(* Logix 5000 project; controller Carpenter_Meter_SCP vendor 1 type 14 code 217 rev 31.11; software revision 31.01; part 5 of 7 *)
(* tags used below, declared in another part *)
   Carpenter_to_Pawnee_OK : BOOL;   // Carpenter to Pawnee Flow Path Permissive
   CC_HI_8800 : BOOL;   // Meter Skid MS-8800 Intrusion Deactivate Switch to OCC
   CC_HI_8840 : BOOL;   // Meter Skid MS-8840 Intrusion Deactivate Switch to OCC
   CC_OCC_HB : DINT;   // Heartbeat from OCC to SCP
   CC_PI_1101 : OCC_Analog;   // Station Discharge Pressure to OCC
   CC_SCP_HB : DINT;   // Heartbeat from SCP to OCC
   CC_XA_0020A : BOOL;   // SCP Main Panel 24VDC Fail to OCC
   CC_XA_0021A : BOOL;   // FGP Main Panel 24VDC Fail to OCC
   CC_XI_0001 : BOOL;   // QA Building Intrusion Deactivate Switch to OCC
   CC_XI_0001A : BOOL;   // QA Building Intrusion Switch to OCC
   CC_XI_0011A : BOOL;   // PDC Building Intrusion Switch to OCC
   CC_XI_0011B : BOOL;   // PDC Building Intrusion Deactivate Switch to OCC
   CC_XI_0020 : BOOL;   // SCP Main PLC 24VDC Failure to OCC
   CC_XI_8800 : BOOL;   // Meter Skid MS-8800 Intrusion Switch to OCC
   CC_XI_8800A : BOOL;   // MS8800 SCP 24VDC Failure to OCC
   CC_XI_8840 : BOOL;   // Meter Skid MS-8840 Intrusion Switch to OCC
   CC_XI_8840A : BOOL;   // MS8840 SCP 24VDC Failure to OCC
   CC_ZI_1100A : BOOL;   // Pig Launched Pig Sig to OCC
   CC_ZI_1100B : BOOL;   // Pig Station Depart Pig Sig to OCC
   CCS_AI_0001 : OCC_Analog;   // QA Building Gas Detector to OCC (AIT-0001)
   CCS_AI_8800A : OCC_Analog;   // Meter Skid MS-8800 Gas Detector #1 (AIT-8800A)
   CCS_AI_8800B : OCC_Analog;   // Meter Skid MS-8800 Gas Detector #2 (AIT-8800B)
   CCS_AI_8840A : OCC_Analog;   // Meter Skid MS-8840 Gas Detector #1 (AIT-8840A)
   CCS_AI_8840B : OCC_Analog;   // Meter Skid MS-8840 Gas Detector #2 (AIT-8840B)
   CCS_ESD_Active : BOOL;   // Station ESD Active to OCC
   CCS_ESD_OCC : BOOL;   // Station ESD Command from OCC
   CCS_FGP_Deactivate : BOOL;   // Fire and Gas Deactivated Status to OCC
   CCS_HI_0011A : BOOL;   // PDC ESD Pushbutton to OCC
   CCS_HI_0017 : BOOL;   // PDC Building PLC Panel ESD Pushbutton to OCC
   CCS_HI_0112A : BOOL;   // QA Building ESD Pushbutton #1 to OCC
   CCS_HI_0112B : BOOL;   // QA Building ESD Pushbutton #2 to OCC
   CCS_HI_0113 : BOOL;   // South Gate ESD Pushbutton to OCC
   CCS_HI_0114 : BOOL;   // North Gate ESD Pushbutton to OCC
   CCS_HI_8800A : BOOL;   // Meter Skid MS-8800 ESD Pushbutton #1 to OCC
   CCS_HI_8800B : BOOL;   // Meter Skid MS-8800 ESD Pushbutton #2 to OCC
   CCS_HI_8840A : BOOL;   // Meter Skid MS-8840 ESD Pushbutton #1 to OCC
   CCS_HI_8840B : BOOL;   // Meter Skid MS-8840 ESD Pushbutton #1 to OCC
   CCS_LAH_3000 : BOOL;   // Sump Tank TU-3000 Leak Detection Switch to OCC
   CCS_LAH_3000_inhibit : BOOL;   // Sump Tank TU-3000 Leak Detection Switch Inhibited to OCC
   CCS_LAH_3100 : BOOL;   // Sump Tank TU-3100 Leak Detection Switch to OCC
   CCS_LAH_3100_inhibit : BOOL;   // Sump Tank TU-3100 Leak Detection Switch Inhibited to OCC
   CCS_LAHH_3000 : BOOL;   // Sump Tank TU-3000 HiHi Level Switch to OCC
   CCS_LAHH_3000_inhibit : BOOL;   // Sump Tank TU-3000 HiHi Level Switch Inhibited to OCC
   CCS_LAHH_3100 : BOOL;   // Sump Tank TU-3100 HiHi Level Switch to OCC
   CCS_LAHH_3100_inhibit : BOOL;   // Sump Tank TU-3100 HiHi Level Switch inhibited to OCC
   CCS_LI_3000 : OCC_Analog;   // Sump Tank TU-3000 Level to OCC
   CCS_LI_3100 : OCC_Analog;   // Sump Tank TU-3000 Level to OCC
   CCS_TI_8010 : OCC_Analog;   // PDC Building Temperature (TIT-8010)
   CCS_XI_0029A : BOOL;   // QA Building Smoke Detector #1 to OCC
   CCS_XI_0029A_Inhibit : BOOL;   // QA Building Smoke Detector #1 Inhibit to OCC
   CCS_XI_0029B : BOOL;   // QA Building Smoke Detector #2 to OCC
   CCS_XI_0029B_Inhibit : BOOL;   // QA Building Smoke Detector #2 Inhibit to OCC
   CCS_XV_0001 : BaseVLVLiquid;   // XV-0001 OCC
   CCS_XV_0041 : BaseVLVLiquid;   // XV-0041 OCC
   CCS_XV_1100 : BaseVLVLiquid;   // XV-1100 OCC
   CCS_XV_1101 : BaseVLVLiquid;   // XV-1101 OCC
   CCS_YI_0022A : BOOL;   // PDC Smoke Detector to OCC
   CCS_YI_0022A_Inhibit : BOOL;   // PDC Smoke Detector Inhibit to OCC
   Cust1_WIOM_Alarm : BOOL;   // Customer 1 WIOM Alarm
   Customer1_Flowpath_OK : BOOL;   // Customer #1 Flowpath Permissive (1 = OK)
   Customer5_Flowpath_OK : BOOL;   // Customer #5 Flowpath Permissive (1 = OK)
   fgp_deactivate_keysw : BOOL;   // Fire and Gas System Deactivated through Key Switch
   FGP_ESD : TGE_Alarm;   // ESD Shutdown from FGP (HS-0020A)
   FGP_Produced : BasProdCons;   // FGP Produced Data
   FGP_SCADA : BasProdCons;
   FI_8800 : REAL;   // Meter Skid MS-8800 Flow Rate in GSV from EFM
   FI_8840 : REAL;   // Meter Skid MS-8840 Flow Rate from EFM
   hb_fail_scada : BOOL;   // SCADA HB Failure
   hb_timer_scada : TIMER;   // SCADA HB Timer
   Launcher_Pig_Sig : TGE_Alarm;   // Launcher Pig Signal (ZS-1100A)
   Main_FGP_24VDC_Fail : TGE_Alarm;   // Main PLC FGP 24VDC Fail (XS-0021)
   MS8800_Biocide_BBL_Per_Day : REAL;   // MS8800 Biocide Flow Rate in BBL/Day (Based off set target of 500PPM)
   MS8800_Biocide_Flow_SP : REAL;   // Meter Skid MS-8800 Biocide Flow Rate Gal/Day
   MS8800_Biocide_RunReq : BOOL;   // Meter Skid MS8800 Biocide Run Req
   MS8800_Cust_Press : TGE_AI_UDT;   // Meter Skid MS-8800 Customer Inlet Pressure (Communicated from Cust)
   MS8800_Flow_Control : PID;   // Meter Skid MS8800 Flow Rate P&ID
   MS8800_Inlet_Press_Control : PID;   // Meter Skid MS8800 Customer Inlet Pressure P&ID
   MS8800_Intrusion : IntrusionAlm;   // Meter Skid MS-8800 Intrusion #1 Alarm
   MS8800_OilFlow_BBL_Per_Day : REAL;   // Meter Skid MS-8800 Oil Flow Rate in BBL/Day
   MS8800_PCV_Pos_AOI : TGE_AI;   // Meter Skid MS-8800 Pressure Control Valve - Position Feedback (PCV-0001)
   MS8800_WaterFlow_BBL_Per_Day : REAL;   // MS8800 Water Flow Rate in BBL/Day (Based off 1% oil in water)
   MS8840_Biocide_BBL_Per_Day : REAL;   // MS8840 Biocide Flow Rate in BBL/Day (Based off set target of 500PPM)
   MS8840_Biocide_Flow_SP : REAL;   // Meter Skid MS-8840 Biocide Flow Rate Gal/Day
   MS8840_Biocide_RunReq : BOOL;   // Meter Skid MS8840 Biocide Run Req
   MS8840_Cust_Press : TGE_AI_UDT;   // Meter Skid MS-8840 Customer Inlet Pressure (Communicated from Cust)
   MS8840_Flow_Control : PID;   // Meter Skid MS8840 Flow Rate P&ID
   MS8840_Inlet_Press_Control : PID;   // Meter Skid MS8840 Customer Inlet Pressure P&ID
   MS8840_Intrusion : IntrusionAlm;   // Meter Skid MS-8840 Intrusion Alarm
   MS8840_OilFlow_BBL_Per_Day : REAL;   // Meter Skid MS-8840 Oil Flow Rate in BBL/Day
   MS8840_PCV_Pos_AOI : TGE_AI;   // Meter Skid MS-8840 Pressure Control Valve - Position Feedback (PCV-0041)
   MS8840_WaterFlow_BBL_Per_Day : REAL;   // MS8840 Water Flow Rate in BBL/Day (Based off 1% oil in water)
   OCC_hb_old : DINT;   // Old OCC HB for diagnostic purposes
   PDC_Bldg_Intrusion : IntrusionAlm;   // PDC Building Intrusion Alarm
   PIC_0001A_Out : REAL;   // Control Valve Output Variable Related to Inlet Pressure
   PIC_0001B_Out : REAL;   // Control Valve Ouptut Variable related to Flow Rate
   PIC_0041A_Out : REAL;   // Control Valve Output Variable Related to Inlet Pressure
   PIC_0041B_Out : REAL;   // Control Valve Ouptut Variable related to Flow Rate
   PV0001_Error : REAL;   // PV0001 Command vs. Feedback Error
   PV0001_Malf : TGE_Alarm;   // PV0001 Malfunction Alarm
   PV0001_Pos_Cmd : REAL;   // PCV-0001 Position Command
   PV0041_Error : REAL;   // PV0041 Command vs. Feedback Error
   PV0041_Malf : TGE_Alarm;   // PV0041 Malfunction Alarm
   PV0041_Pos_Cmd : REAL;   // PCV-0041 Position Command
   pv_0001_pid_tmr : TIMER;
   pv_0041_pid_tmr : TIMER;
   QA_Bldg_Intrusion : IntrusionAlm;   // QA Building Intrusion Alarm Bit 0-7 = Bldg Int Switch Bit 15 = Deact HS
   SCP_Produced : BasProdCons;
   Sta_Stat : StaStatus;
   sta_stop_vlv_req : BOOL;   // Station Stop Valve Close Request
   Station_Depart_Pig_Sig : TGE_Alarm;   // Station Departed Pig Signal (ZS-1100B)
   Station_Disch_Press : TGE_AI_UDT;   // Station Discharge Pressure - Launcher Skid (PIT-1101)
   TU3000_HiHi_Lvl : TGE_Alarm;   // Sump Tank (TU-3000) Hi Hi Level Switch (LSHH-3000)
   TU3000_Leak_Detect : TGE_Alarm;   // Sump Tank (TU-3000) Leak Detected (LSH-3000)
   TU3000_Level : TGE_AI_UDT;   // Sump Tank (TU-3000) Level Transmitter (LIT-3000)
   TU3100_HiHi_Lvl : TGE_Alarm;   // Sump Tank (TU-3100) Hi Hi Level Switch (LSHH-3100)
   TU3100_Leak_Detect : TGE_Alarm;   // Sump Tank (TU-3100) Leak Detected (LSH-3100)
   TU3100_Level : TGE_AI_UDT;   // Sump Tank (TU-3100) Level Transmitter (LIT-3100)
   watchdog_tmr : TIMER;   // Watchdog Timer for Communications
   XV_0001 : BaseVLVLiquid;   // XV-0001
   XV_0041 : BaseVLVLiquid;   // XV-0041
   XV_1100 : BaseVLVLiquid;   // XV-1100
   XV_1101 : BaseVLVLiquid;   // XV-1101
(* Map_Inputs, continued *)

ROUTINE Main   (* ladder *)
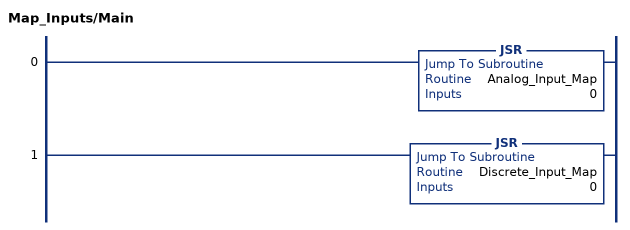
   0: JSR(Analog_Input_Map,0);
   1: JSR(Discrete_Input_Map,0);
END_ROUTINE
END_PROGRAM

PROGRAM Map_Outputs   (* main routine Main *)

ROUTINE Analog_Output_Map   (* ladder *)
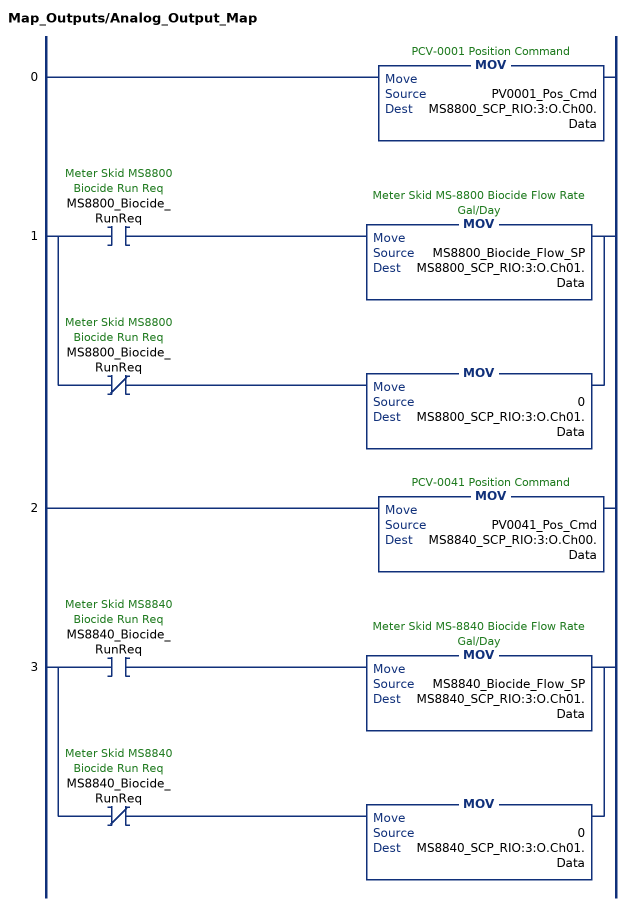
   0: MOV(PV0001_Pos_Cmd,MS8800_SCP_RIO:3:O.Ch00.Data);
   1: [XIC(MS8800_Biocide_RunReq) MOV(MS8800_Biocide_Flow_SP,MS8800_SCP_RIO:3:O.Ch01.Data) ,XIO(MS8800_Biocide_RunReq) MOV(0,MS8800_SCP_RIO:3:O.Ch01.Data) ];
   2: MOV(PV0041_Pos_Cmd,MS8840_SCP_RIO:3:O.Ch00.Data);
   3: [XIC(MS8840_Biocide_RunReq) MOV(MS8840_Biocide_Flow_SP,MS8840_SCP_RIO:3:O.Ch01.Data) ,XIO(MS8840_Biocide_RunReq) MOV(0,MS8840_SCP_RIO:3:O.Ch01.Data) ];
END_ROUTINE

ROUTINE Discrete_Output_Map   (* ladder *)
   0: NOP();
END_ROUTINE

ROUTINE Main   (* ladder *)
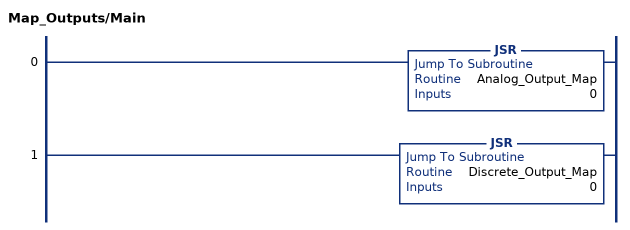
   0: JSR(Analog_Output_Map,0);
   1: JSR(Discrete_Output_Map,0);
END_ROUTINE
END_PROGRAM

PROGRAM Meter_Skid_Control   (* main routine Main *)

ROUTINE Main   (* ladder *)
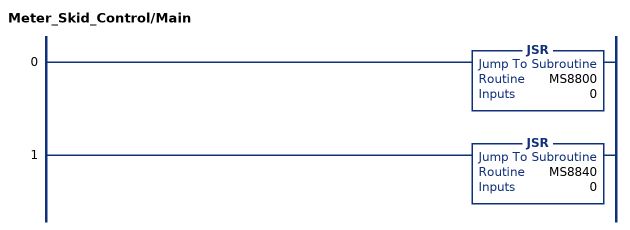
   0: JSR(MS8800,0);
   1: JSR(MS8840,0);
END_ROUTINE

ROUTINE MS8800   (* ladder *)
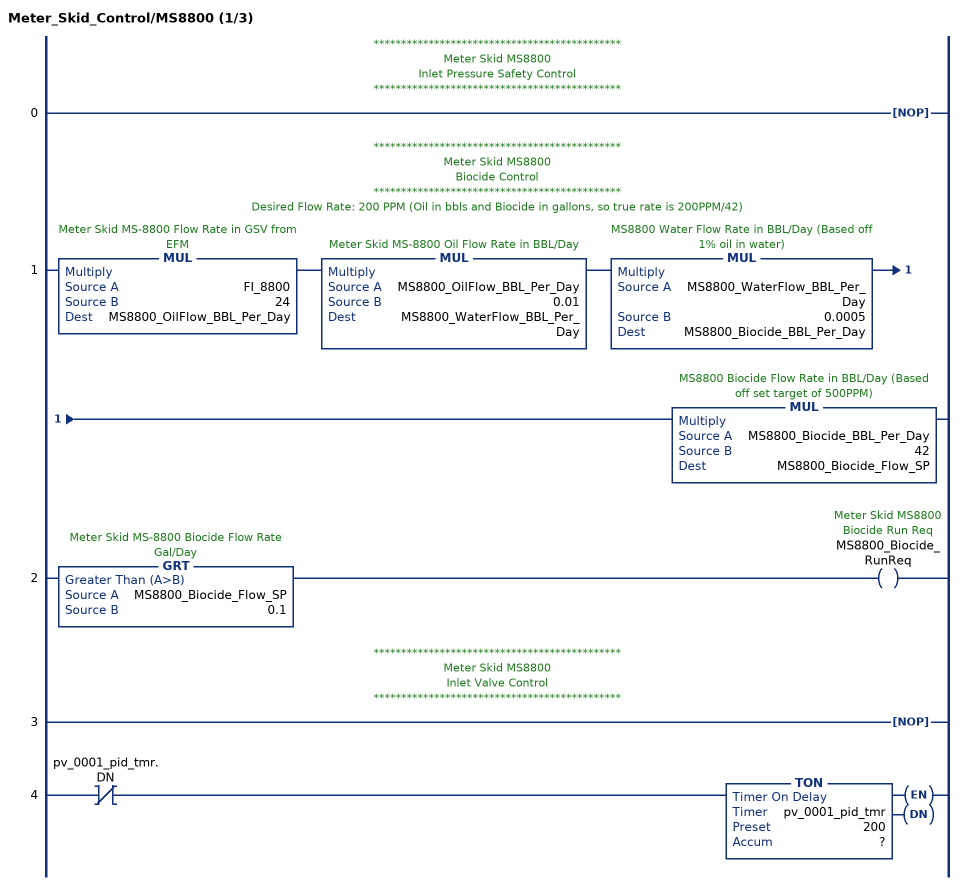
   // *********************************************
   // Meter Skid MS8800
   // Inlet Pressure Safety Control
   // *********************************************
   0: NOP();
   // *********************************************
   // Meter Skid MS8800
   // Biocide Control
   // *********************************************
   // Desired Flow Rate: 200 PPM (Oil in bbls and Biocide in gallons, so true rate is 200PPM/42)
   1: MUL(FI_8800,24,MS8800_OilFlow_BBL_Per_Day)MUL(MS8800_OilFlow_BBL_Per_Day,0.01,MS8800_WaterFlow_BBL_Per_Day)MUL(MS8800_WaterFlow_BBL_Per_Day,0.0005,MS8800_Biocide_BBL_Per_Day)MUL(MS8800_Biocide_BBL_Per_Day,42,MS8800_Biocide_Flow_SP);
   2: GRT(MS8800_Biocide_Flow_SP,0.1)OTE(MS8800_Biocide_RunReq);
   // *********************************************
   // Meter Skid MS8800
   // Inlet Valve Control
   // *********************************************
   3: NOP();
   4: XIO(pv_0001_pid_tmr.DN)TON(pv_0001_pid_tmr,?,?);
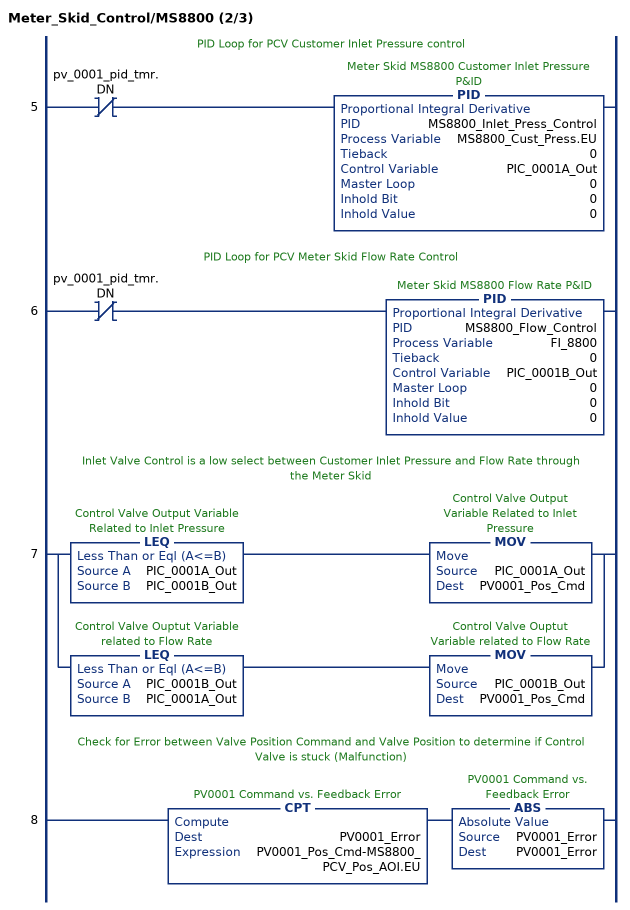
   // PID Loop for PCV Customer Inlet Pressure control
   5: XIO(pv_0001_pid_tmr.DN)PID(MS8800_Inlet_Press_Control,MS8800_Cust_Press.EU,0,PIC_0001A_Out,0,0,0);
   // PID Loop for PCV Meter Skid Flow Rate Control
   6: XIO(pv_0001_pid_tmr.DN)PID(MS8800_Flow_Control,FI_8800,0,PIC_0001B_Out,0,0,0);
   // Inlet Valve Control is a low select between Customer Inlet Pressure and Flow Rate through the Meter Skid
   7: [LEQ(PIC_0001A_Out,PIC_0001B_Out) MOV(PIC_0001A_Out,PV0001_Pos_Cmd) ,LEQ(PIC_0001B_Out,PIC_0001A_Out) MOV(PIC_0001B_Out,PV0001_Pos_Cmd) ];
   // Check for Error between Valve Position Command and Valve Position to determine if Control Valve is stuck (Malfunction)
   8: CPT(PV0001_Error,PV0001_Pos_Cmd-MS8800_PCV_Pos_AOI.EU)ABS(PV0001_Error,PV0001_Error);
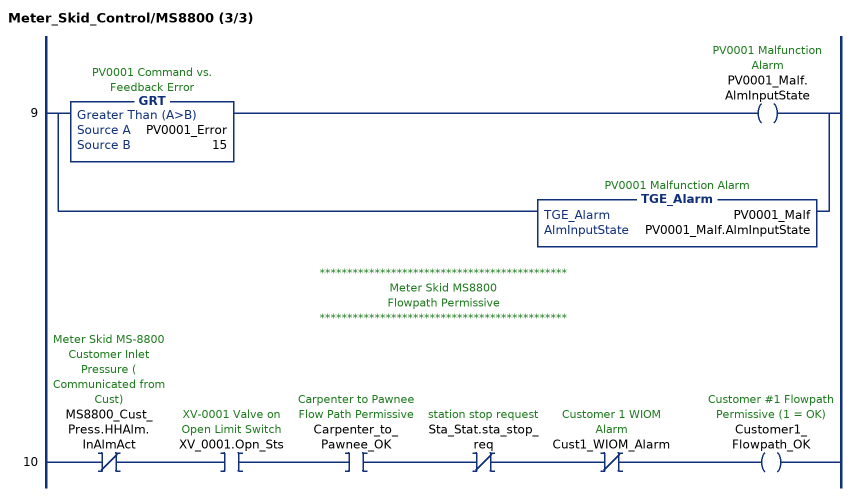
   9: [GRT(PV0001_Error,15) OTE(PV0001_Malf.AlmInputState) ,TGE_Alarm(PV0001_Malf,PV0001_Malf.AlmInputState) ];
   // *********************************************
   // Meter Skid MS8800
   // Flowpath Permissive
   // *********************************************
   10: XIO(MS8800_Cust_Press.HHAlm.InAlmAct)XIC(XV_0001.Opn_Sts)XIC(Carpenter_to_Pawnee_OK)XIO(Sta_Stat.sta_stop_req)XIO(Cust1_WIOM_Alarm)OTE(Customer1_Flowpath_OK);
END_ROUTINE

ROUTINE MS8840   (* ladder *)
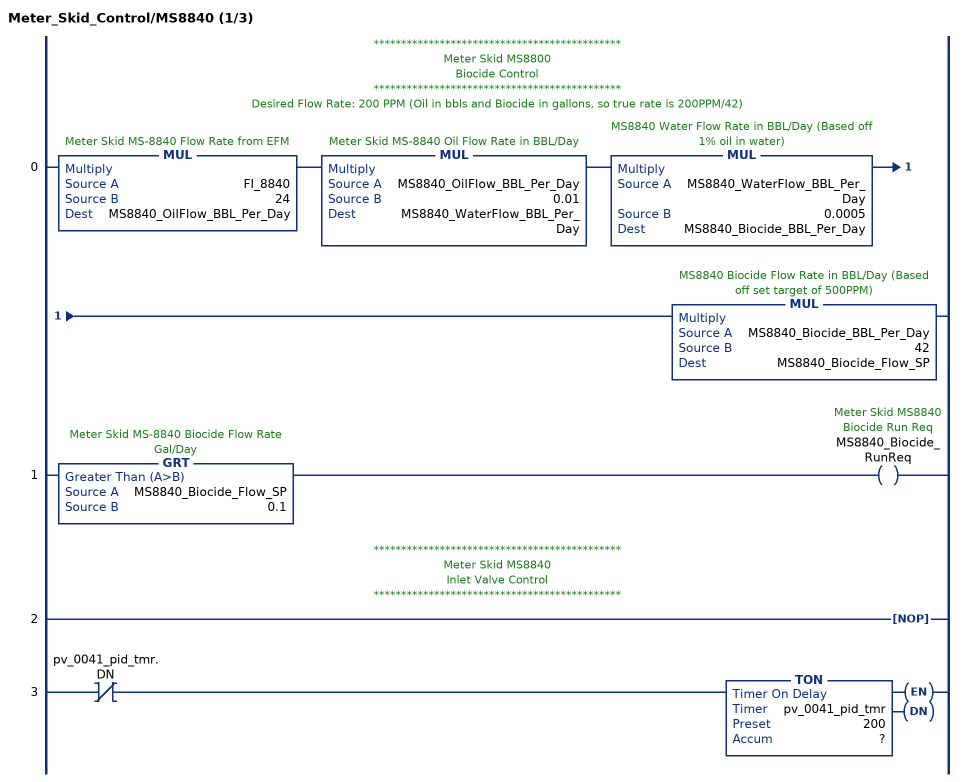
   // *********************************************
   // Meter Skid MS8800
   // Biocide Control
   // *********************************************
   // Desired Flow Rate: 200 PPM (Oil in bbls and Biocide in gallons, so true rate is 200PPM/42)
   0: MUL(FI_8840,24,MS8840_OilFlow_BBL_Per_Day)MUL(MS8840_OilFlow_BBL_Per_Day,0.01,MS8840_WaterFlow_BBL_Per_Day)MUL(MS8840_WaterFlow_BBL_Per_Day,0.0005,MS8840_Biocide_BBL_Per_Day)MUL(MS8840_Biocide_BBL_Per_Day,42,MS8840_Biocide_Flow_SP);
   1: GRT(MS8840_Biocide_Flow_SP,0.1)OTE(MS8840_Biocide_RunReq);
   // *********************************************
   // Meter Skid MS8840
   // Inlet Valve Control
   // *********************************************
   2: NOP();
   3: XIO(pv_0041_pid_tmr.DN)TON(pv_0041_pid_tmr,?,?);
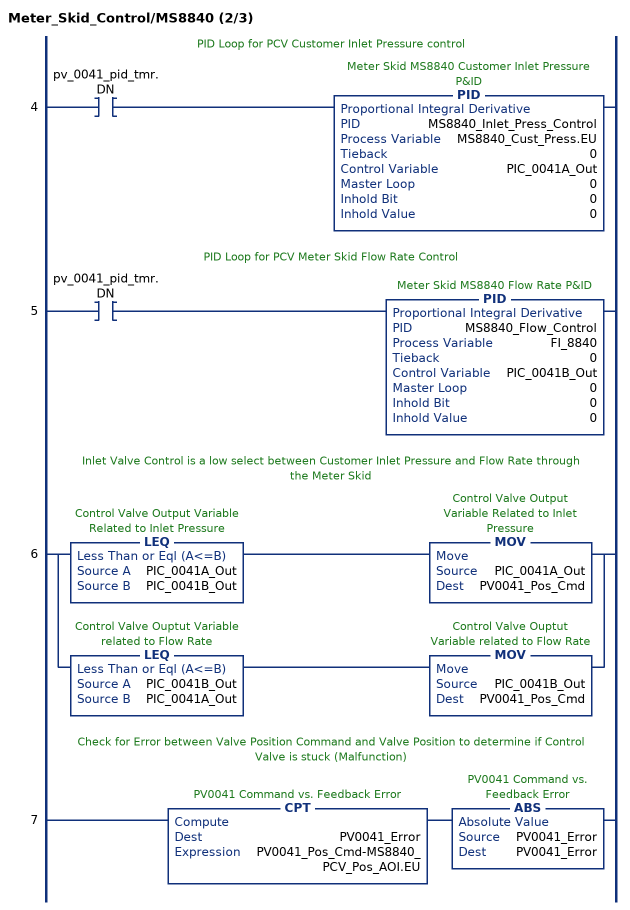
   // PID Loop for PCV Customer Inlet Pressure control
   4: XIC(pv_0041_pid_tmr.DN)PID(MS8840_Inlet_Press_Control,MS8840_Cust_Press.EU,0,PIC_0041A_Out,0,0,0);
   // PID Loop for PCV Meter Skid Flow Rate Control
   5: XIC(pv_0041_pid_tmr.DN)PID(MS8840_Flow_Control,FI_8840,0,PIC_0041B_Out,0,0,0);
   // Inlet Valve Control is a low select between Customer Inlet Pressure and Flow Rate through the Meter Skid
   6: [LEQ(PIC_0041A_Out,PIC_0041B_Out) MOV(PIC_0041A_Out,PV0041_Pos_Cmd) ,LEQ(PIC_0041B_Out,PIC_0041A_Out) MOV(PIC_0041B_Out,PV0041_Pos_Cmd) ];
   // Check for Error between Valve Position Command and Valve Position to determine if Control Valve is stuck (Malfunction)
   7: CPT(PV0041_Error,PV0041_Pos_Cmd-MS8840_PCV_Pos_AOI.EU)ABS(PV0041_Error,PV0041_Error);
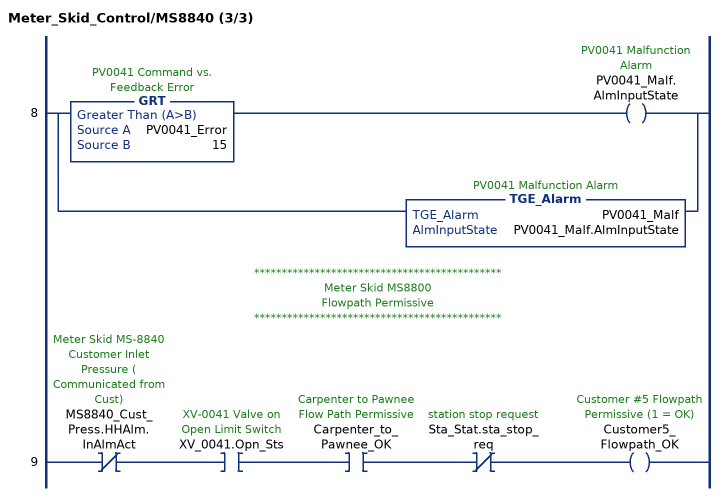
   8: [GRT(PV0041_Error,15) OTE(PV0041_Malf.AlmInputState) ,TGE_Alarm(PV0041_Malf,PV0041_Malf.AlmInputState) ];
   // *********************************************
   // Meter Skid MS8800
   // Flowpath Permissive
   // *********************************************
   9: XIO(MS8840_Cust_Press.HHAlm.InAlmAct)XIC(XV_0041.Opn_Sts)XIC(Carpenter_to_Pawnee_OK)XIO(Sta_Stat.sta_stop_req)OTE(Customer5_Flowpath_OK);
END_ROUTINE
END_PROGRAM

PROGRAM OCC_Comms   (* main routine OCC_Comms_Main *)

ROUTINE OCC_Comms_Main   (* ladder *)
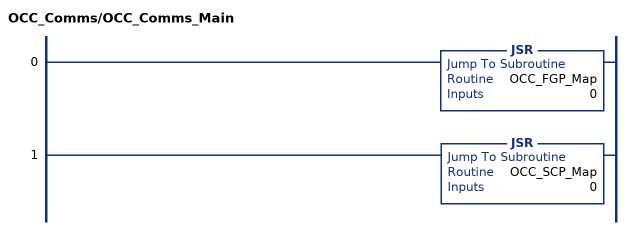
   0: JSR(OCC_FGP_Map,0);
   1: JSR(OCC_SCP_Map,0);
END_ROUTINE

ROUTINE OCC_FGP_Map   (* ladder *)
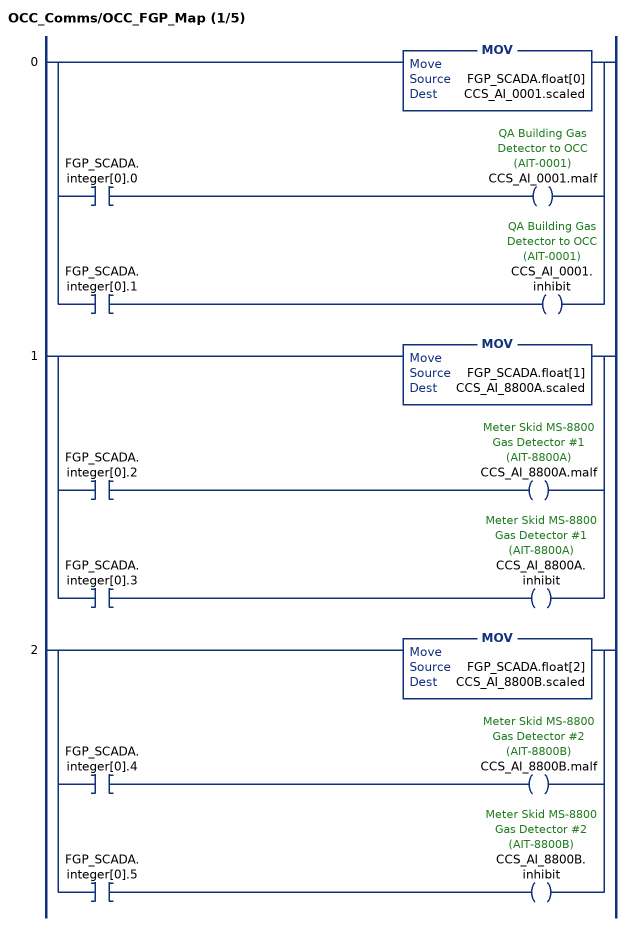
   0: [MOV(FGP_SCADA.float[0],CCS_AI_0001.scaled) ,XIC(FGP_SCADA.integer[0].0) OTE(CCS_AI_0001.malf) ,XIC(FGP_SCADA.integer[0].1) OTE(CCS_AI_0001.inhibit) ];
   1: [MOV(FGP_SCADA.float[1],CCS_AI_8800A.scaled) ,XIC(FGP_SCADA.integer[0].2) OTE(CCS_AI_8800A.malf) ,XIC(FGP_SCADA.integer[0].3) OTE(CCS_AI_8800A.inhibit) ];
   2: [MOV(FGP_SCADA.float[2],CCS_AI_8800B.scaled) ,XIC(FGP_SCADA.integer[0].4) OTE(CCS_AI_8800B.malf) ,XIC(FGP_SCADA.integer[0].5) OTE(CCS_AI_8800B.inhibit) ];
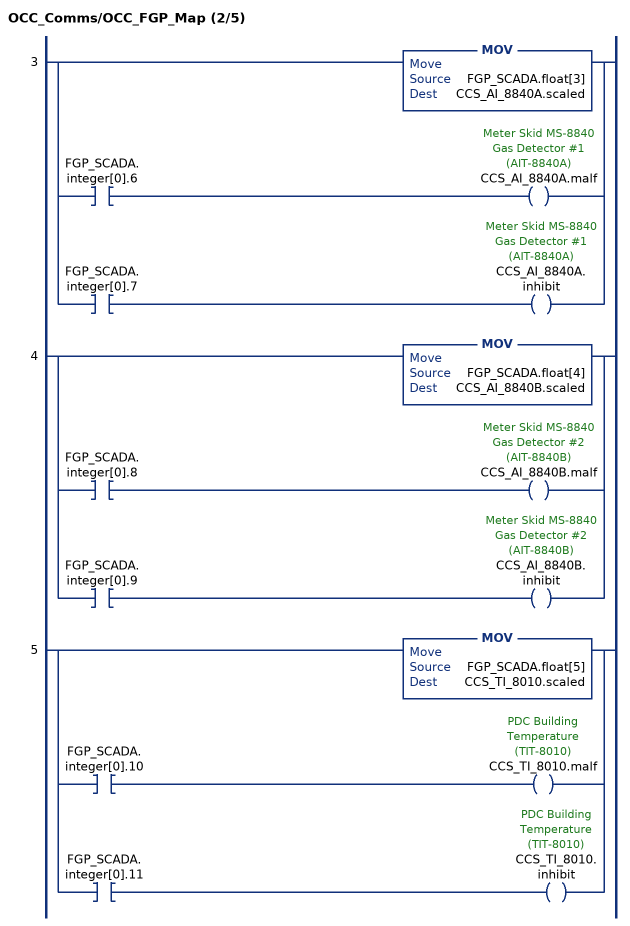
   3: [MOV(FGP_SCADA.float[3],CCS_AI_8840A.scaled) ,XIC(FGP_SCADA.integer[0].6) OTE(CCS_AI_8840A.malf) ,XIC(FGP_SCADA.integer[0].7) OTE(CCS_AI_8840A.inhibit) ];
   4: [MOV(FGP_SCADA.float[4],CCS_AI_8840B.scaled) ,XIC(FGP_SCADA.integer[0].8) OTE(CCS_AI_8840B.malf) ,XIC(FGP_SCADA.integer[0].9) OTE(CCS_AI_8840B.inhibit) ];
   5: [MOV(FGP_SCADA.float[5],CCS_TI_8010.scaled) ,XIC(FGP_SCADA.integer[0].10) OTE(CCS_TI_8010.malf) ,XIC(FGP_SCADA.integer[0].11) OTE(CCS_TI_8010.inhibit) ];
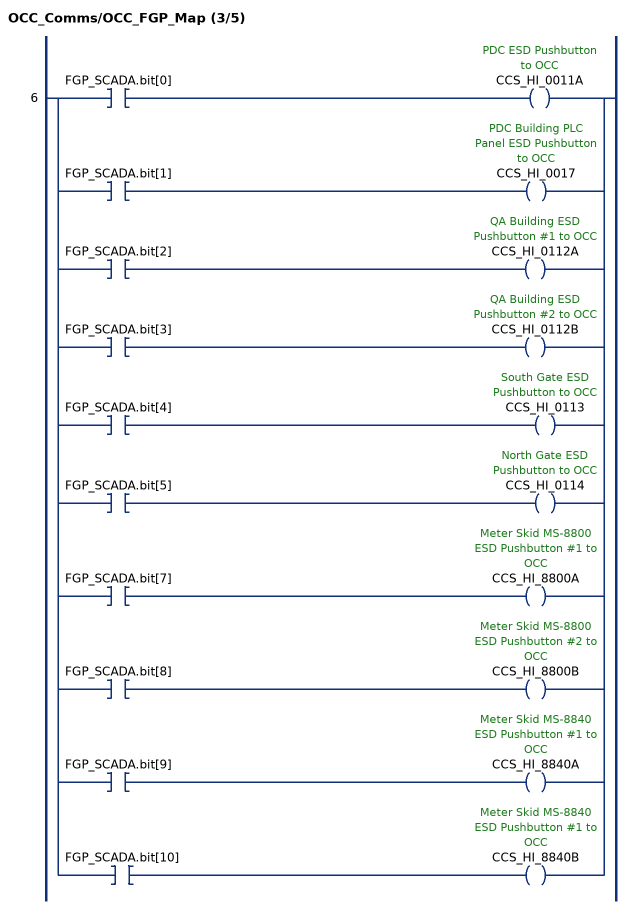
   6: [XIC(FGP_SCADA.bit[0]) OTE(CCS_HI_0011A) ,XIC(FGP_SCADA.bit[1]) OTE(CCS_HI_0017) ,XIC(FGP_SCADA.bit[2]) OTE(CCS_HI_0112A) ,XIC(FGP_SCADA.bit[3]) OTE(CCS_HI_0112B) ,XIC(FGP_SCADA.bit[4]) OTE(CCS_HI_0113) ,XIC(FGP_SCADA.bit[5]) OTE(CCS_HI_0114) ,XIC(FGP_SCADA.bit[7]) OTE(CCS_HI_8800A) ,XIC(FGP_SCADA.bit[8]) OTE(CCS_HI_8800B) ,XIC(FGP_SCADA.bit[9]) OTE(CCS_HI_8840A) ,XIC(FGP_SCADA.bit[10]) OTE(CCS_HI_8840B) ];
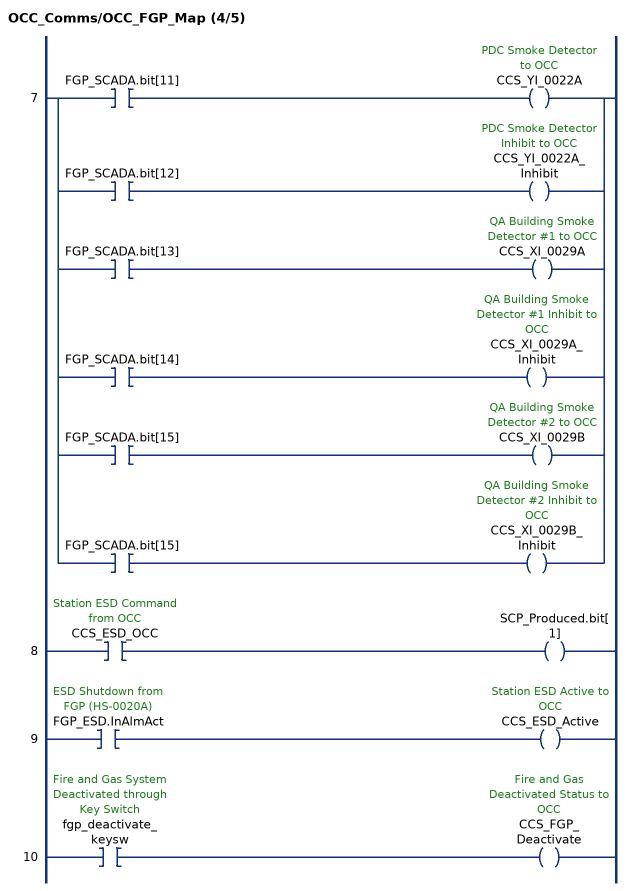
   7: [XIC(FGP_SCADA.bit[11]) OTE(CCS_YI_0022A) ,XIC(FGP_SCADA.bit[12]) OTE(CCS_YI_0022A_Inhibit) ,XIC(FGP_SCADA.bit[13]) OTE(CCS_XI_0029A) ,XIC(FGP_SCADA.bit[14]) OTE(CCS_XI_0029A_Inhibit) ,XIC(FGP_SCADA.bit[15]) OTE(CCS_XI_0029B) ,XIC(FGP_SCADA.bit[15]) OTE(CCS_XI_0029B_Inhibit) ];
   8: XIC(CCS_ESD_OCC)OTE(SCP_Produced.bit[1]);
   9: XIC(FGP_ESD.InAlmAct)OTE(CCS_ESD_Active);
   10: XIC(fgp_deactivate_keysw)OTE(CCS_FGP_Deactivate);
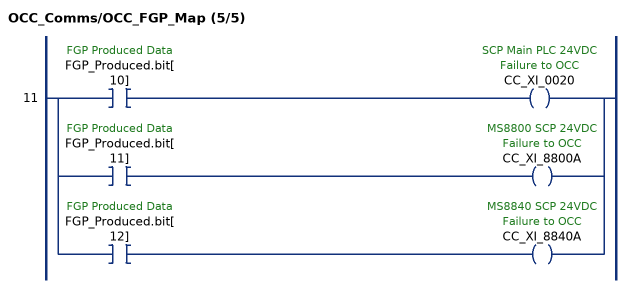
   11: [XIC(FGP_Produced.bit[10]) OTE(CC_XI_0020) ,XIC(FGP_Produced.bit[11]) OTE(CC_XI_8800A) ,XIC(FGP_Produced.bit[12]) OTE(CC_XI_8840A) ];
END_ROUTINE

ROUTINE OCC_SCP_Map   (* ladder *)
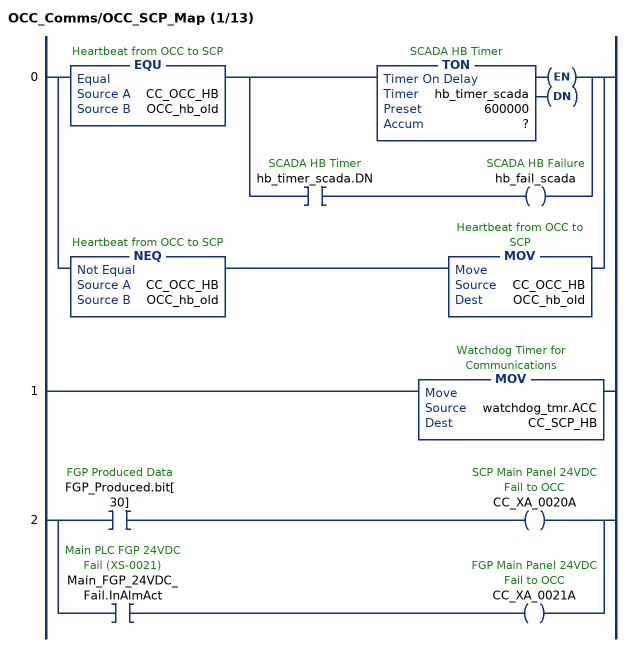
   0: [EQU(CC_OCC_HB,OCC_hb_old) [TON(hb_timer_scada,?,?) ,XIC(hb_timer_scada.DN) OTE(hb_fail_scada) ] ,NEQ(CC_OCC_HB,OCC_hb_old) MOV(CC_OCC_HB,OCC_hb_old) ];
   1: MOV(watchdog_tmr.ACC,CC_SCP_HB);
   2: [XIC(FGP_Produced.bit[30]) OTE(CC_XA_0020A) ,XIC(Main_FGP_24VDC_Fail.InAlmAct) OTE(CC_XA_0021A) ];
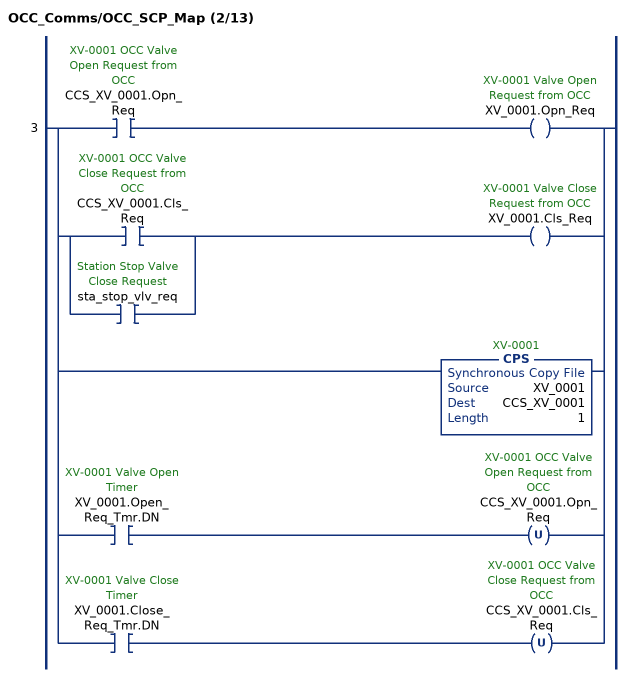
   3: [XIC(CCS_XV_0001.Opn_Req) OTE(XV_0001.Opn_Req) ,[XIC(CCS_XV_0001.Cls_Req) ,XIC(sta_stop_vlv_req) ] OTE(XV_0001.Cls_Req) ,CPS(XV_0001,CCS_XV_0001,1) ,XIC(XV_0001.Open_Req_Tmr.DN) OTU(CCS_XV_0001.Opn_Req) ,XIC(XV_0001.Close_Req_Tmr.DN) OTU(CCS_XV_0001.Cls_Req) ];
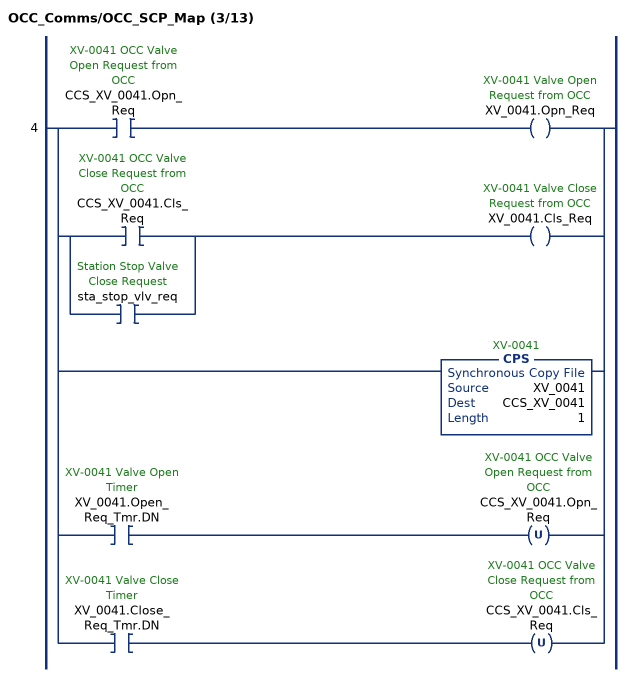
   4: [XIC(CCS_XV_0041.Opn_Req) OTE(XV_0041.Opn_Req) ,[XIC(CCS_XV_0041.Cls_Req) ,XIC(sta_stop_vlv_req) ] OTE(XV_0041.Cls_Req) ,CPS(XV_0041,CCS_XV_0041,1) ,XIC(XV_0041.Open_Req_Tmr.DN) OTU(CCS_XV_0041.Opn_Req) ,XIC(XV_0041.Close_Req_Tmr.DN) OTU(CCS_XV_0041.Cls_Req) ];
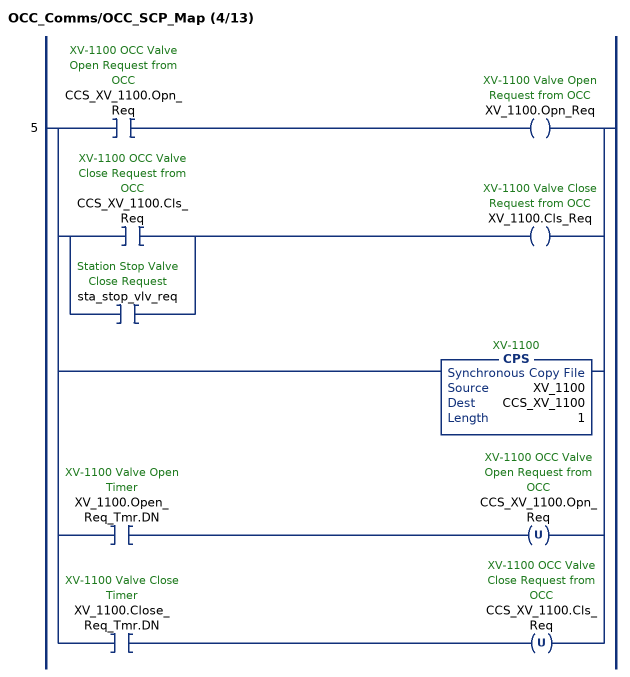
   5: [XIC(CCS_XV_1100.Opn_Req) OTE(XV_1100.Opn_Req) ,[XIC(CCS_XV_1100.Cls_Req) ,XIC(sta_stop_vlv_req) ] OTE(XV_1100.Cls_Req) ,CPS(XV_1100,CCS_XV_1100,1) ,XIC(XV_1100.Open_Req_Tmr.DN) OTU(CCS_XV_1100.Opn_Req) ,XIC(XV_1100.Close_Req_Tmr.DN) OTU(CCS_XV_1100.Cls_Req) ];
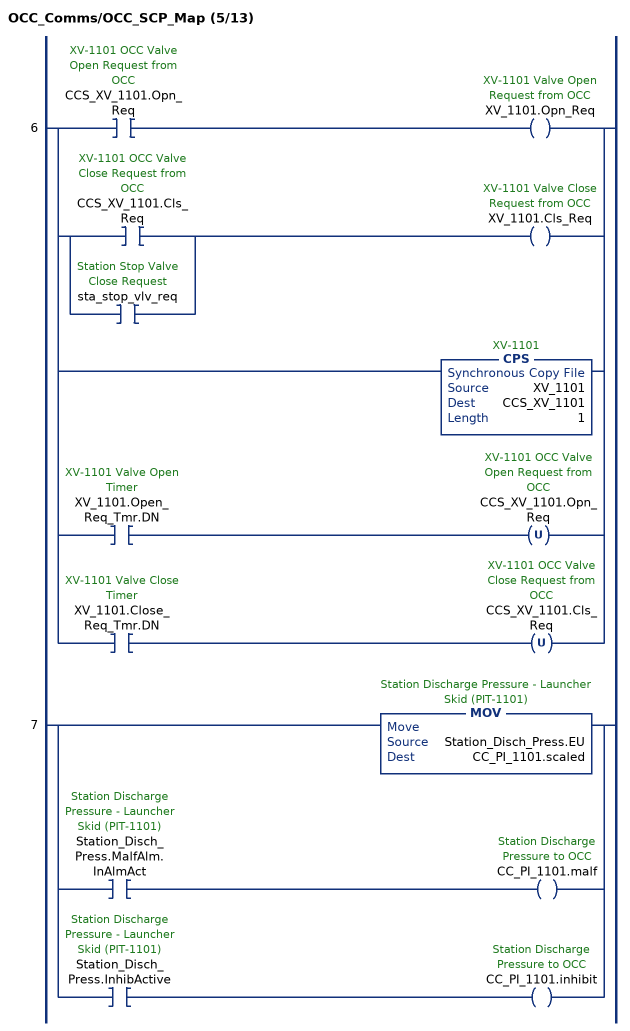
   6: [XIC(CCS_XV_1101.Opn_Req) OTE(XV_1101.Opn_Req) ,[XIC(CCS_XV_1101.Cls_Req) ,XIC(sta_stop_vlv_req) ] OTE(XV_1101.Cls_Req) ,CPS(XV_1101,CCS_XV_1101,1) ,XIC(XV_1101.Open_Req_Tmr.DN) OTU(CCS_XV_1101.Opn_Req) ,XIC(XV_1101.Close_Req_Tmr.DN) OTU(CCS_XV_1101.Cls_Req) ];
   7: [MOV(Station_Disch_Press.EU,CC_PI_1101.scaled) ,XIC(Station_Disch_Press.MalfAlm.InAlmAct) OTE(CC_PI_1101.malf) ,XIC(Station_Disch_Press.InhibActive) OTE(CC_PI_1101.inhibit) ];
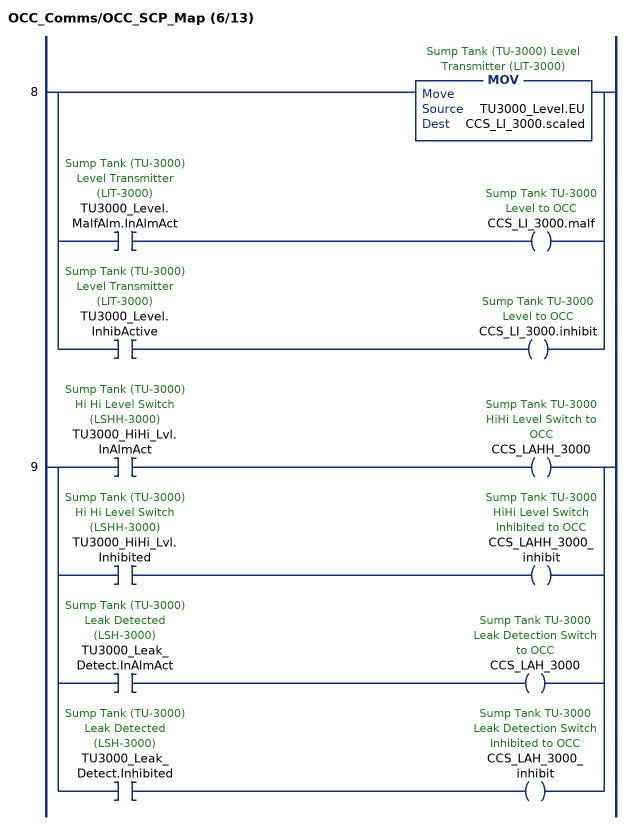
   8: [MOV(TU3000_Level.EU,CCS_LI_3000.scaled) ,XIC(TU3000_Level.MalfAlm.InAlmAct) OTE(CCS_LI_3000.malf) ,XIC(TU3000_Level.InhibActive) OTE(CCS_LI_3000.inhibit) ];
   9: [XIC(TU3000_HiHi_Lvl.InAlmAct) OTE(CCS_LAHH_3000) ,XIC(TU3000_HiHi_Lvl.Inhibited) OTE(CCS_LAHH_3000_inhibit) ,XIC(TU3000_Leak_Detect.InAlmAct) OTE(CCS_LAH_3000) ,XIC(TU3000_Leak_Detect.Inhibited) OTE(CCS_LAH_3000_inhibit) ];
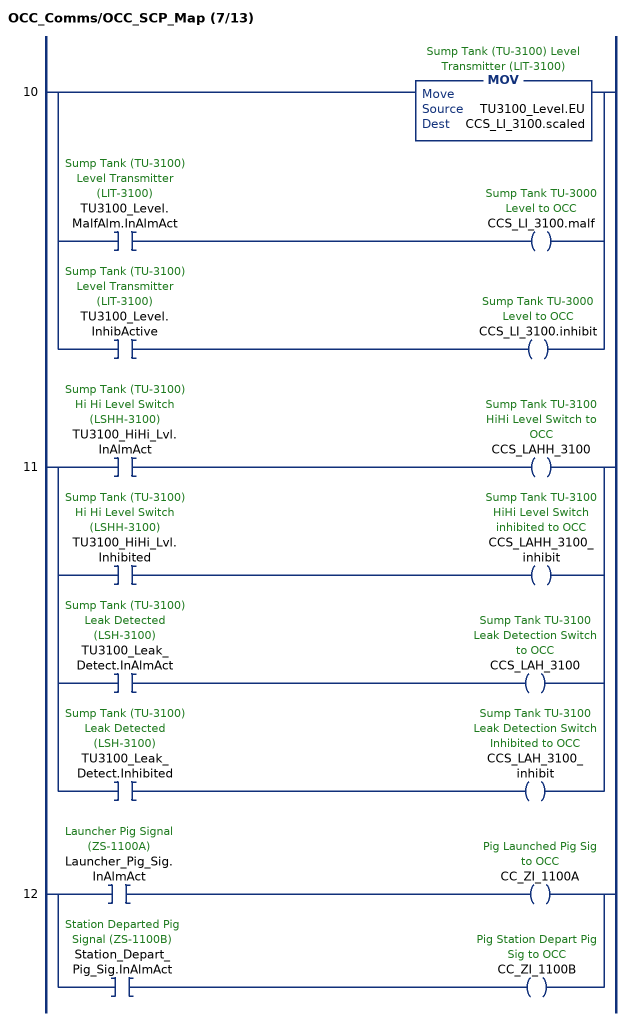
   10: [MOV(TU3100_Level.EU,CCS_LI_3100.scaled) ,XIC(TU3100_Level.MalfAlm.InAlmAct) OTE(CCS_LI_3100.malf) ,XIC(TU3100_Level.InhibActive) OTE(CCS_LI_3100.inhibit) ];
   11: [XIC(TU3100_HiHi_Lvl.InAlmAct) OTE(CCS_LAHH_3100) ,XIC(TU3100_HiHi_Lvl.Inhibited) OTE(CCS_LAHH_3100_inhibit) ,XIC(TU3100_Leak_Detect.InAlmAct) OTE(CCS_LAH_3100) ,XIC(TU3100_Leak_Detect.Inhibited) OTE(CCS_LAH_3100_inhibit) ];
   12: [XIC(Launcher_Pig_Sig.InAlmAct) OTE(CC_ZI_1100A) ,XIC(Station_Depart_Pig_Sig.InAlmAct) OTE(CC_ZI_1100B) ];
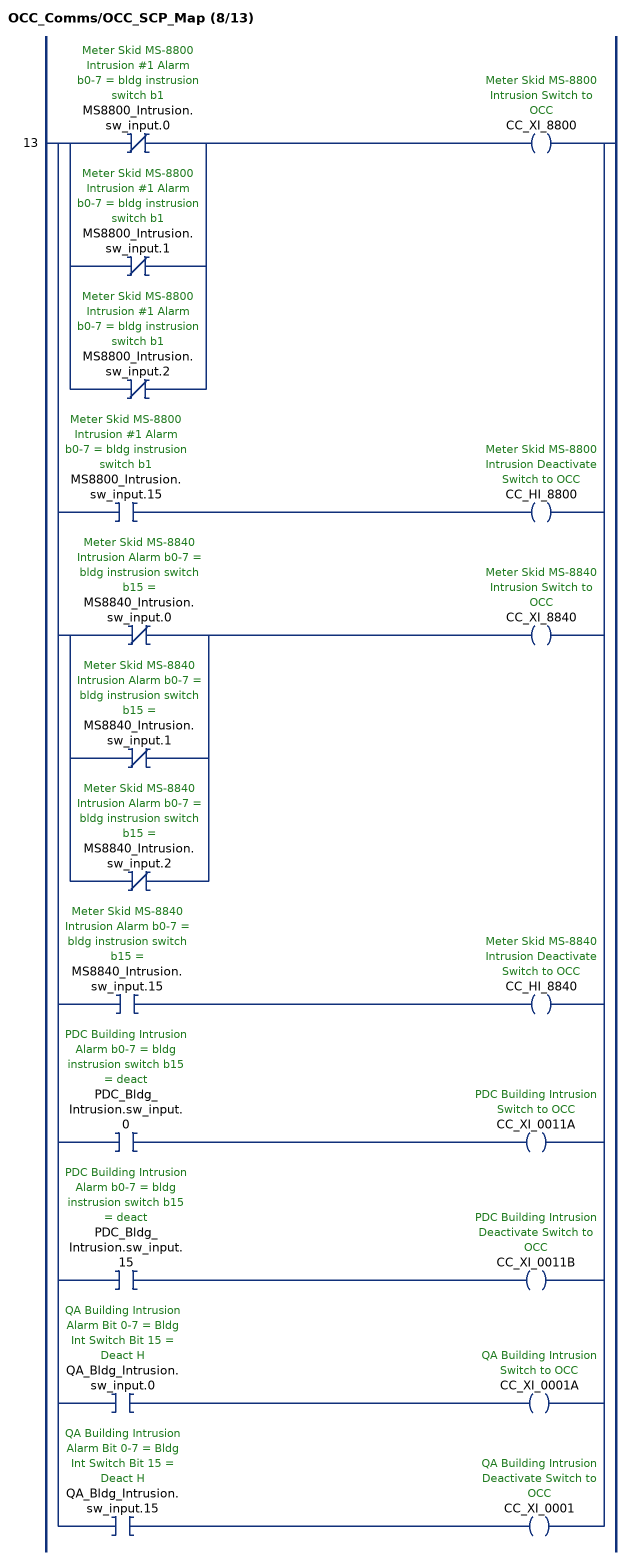
   13: [[XIO(MS8800_Intrusion.sw_input.0) ,XIO(MS8800_Intrusion.sw_input.1) ,XIO(MS8800_Intrusion.sw_input.2) ] OTE(CC_XI_8800) ,XIC(MS8800_Intrusion.sw_input.15) OTE(CC_HI_8800) ,[XIO(MS8840_Intrusion.sw_input.0) ,XIO(MS8840_Intrusion.sw_input.1) ,XIO(MS8840_Intrusion.sw_input.2) ] OTE(CC_XI_8840) ,XIC(MS8840_Intrusion.sw_input.15) OTE(CC_HI_8840) ,XIC(PDC_Bldg_Intrusion.sw_input.0) OTE(CC_XI_0011A) ,XIC(PDC_Bldg_Intrusion.sw_input.15) OTE(CC_XI_0011B) ,XIC(QA_Bldg_Intrusion.sw_input.0) OTE(CC_XI_0001A) ,XIC(QA_Bldg_Intrusion.sw_input.15) OTE(CC_XI_0001) ];
